(* PLC project ClaudeUnGuided.project, Rexroth ctrlX PLC Engineering ctrlX PLC 4.6.2 *)
(* stored: creationDateTime 2026-10-09T23:50:41.8125568, modificationDateTime 2026-10-09T23:34:18.6487849 *)

PROGRAM OtherOperators
  VAR
    bChoice : BOOL;
    In1 : INT;
    In2 : INT;
    out1 : INT;
    iMuxSel : INT;
    in3 : INT;
    in4 : INT;
    in5 : INT;
    out2 : INT;
    minVal : INT;
    maxVal : INT;
    out3 : INT;
    out4 : REAL;
  END_VAR

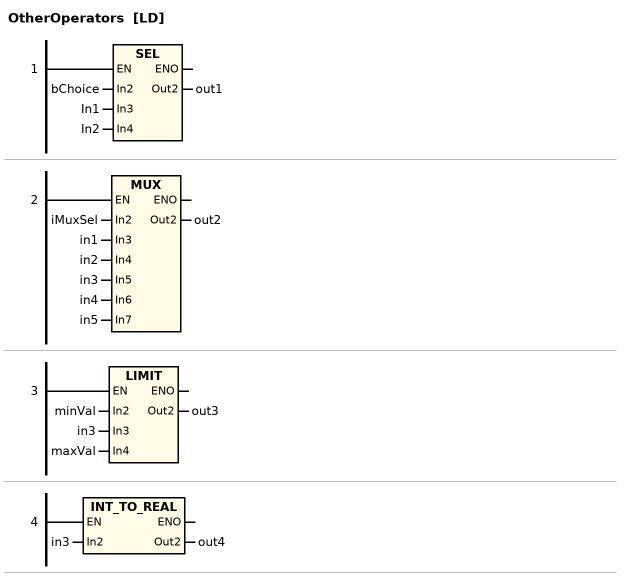
(* LD diagram, written out as Structured Text *)
(* --- network: Select --- *)
out1 := SEL(In2 := bChoice, In3 := In1, In4 := In2);

out2 := MUX(In2 := iMuxSel, In3 := in1, In4 := in2, In5 := in3, In6 := in4, In7 := in5);

out3 := LIMIT(In2 := minVal, In3 := in3, In4 := maxVal);

out4 := INT_TO_REAL(In2 := in3);
END_PROGRAM
